// TIA Portal V20 export
FUNCTION_BLOCK "FB_HmiKeysSignalsManu"   // FB813, SCL
{ S7_Optimized_Access := 'TRUE' }
// stored: AutoNumber false, MemoryReserve 100, SetENOAutomatically false
   VAR_IN_OUT
      ioOPC : "UDT_OPC_Button";
   END_VAR
   VAR
      sKeySWStatus : Bool;
      sKeySWToggleStatus : Bool;
      sKeyDisable : Bool;
      sKeySWPositiveFront : Bool;
      sKeySWNegativeFront : Bool;
      sKeySWTogglePositiveFront : Bool;
      sKeySWToggleNegativeFront : Bool;
      sLedSWStatus : Bool;
      sLedSWStatusBlink : Bool;
      sRT_KeySWPositiveFront { S7_SetPoint := 'True'} : R_TRIG;
      sFT_KeySWNegativeFront { S7_SetPoint := 'True'} : F_TRIG;
      sRT_KeySWTogglePositiveFront { S7_SetPoint := 'True'} : R_TRIG;
      sFT_KeySWToggleNegativeFront { S7_SetPoint := 'True'} : F_TRIG;
   END_VAR
BEGIN
   REGION Description header 
       //==================================================================================
       // POSALUX Swiss SA / (C) Copyright 2025
       //----------------------------------------------------------------------------------
       // Title: FB_HmiKeysSignalsManu 
       // Comment/Function: 
       //
       // Author: Fabien Waldt
       // Engineering: TIA Portal v19
       //----------------------------------------------------------------------------------
       // Change log table:
       // Version  | Date     | Expert in charge | Changes applied
       // ---------|----------|------------------|------------------------------------
       // 00.00.01 | 20250911 | WFA              | First released version
       // ==================================================================================
   END_REGION

   REGION Key Enable
       #ioOPC.bEnable := NOT #sKeyDisable;
   END_REGION

   REGION Inputs keys
           // Management of the software input
           IF NOT #sKeyDisable THEN
               #sKeySWStatus := #ioOPC.bClick;
           // ELSE
           //     #sKeySWStatus := FALSE;
           //     #sKeySWToggleStatus := FALSE;
           END_IF;

           // Reset KeyOPCStatus (bClick from HMI)
           #ioOPC.bClick := FALSE;

           // Rising/falling edge detection when pressing the button
           #sRT_KeySWPositiveFront(CLK := #sKeySWStatus,
                                  Q => #sKeySWPositiveFront);

           #sFT_KeySWNegativeFront(CLK := #sKeySWStatus,
                                  Q => #sKeySWNegativeFront);

           // Toggle state update
           IF #sKeySWPositiveFront  THEN
               #sKeySWToggleStatus := NOT #sKeySWToggleStatus;
           END_IF;

           // Rising/falling edge detection of the toggle state
           #sRT_KeySWTogglePositiveFront(CLK := #sKeySWToggleStatus,
                                        Q => #sKeySWTogglePositiveFront);

           #sFT_KeySWToggleNegativeFront(CLK := #sKeySWToggleStatus,
                                        Q => #sKeySWToggleNegativeFront);
   END_REGION

   REGION Outputs LED   
       #ioOPC.bIsPressed := TRUE;

       // On / Off Status
       IF #sLedSWStatus THEN
           #ioOPC.eColor := 2;
       ELSE
           #ioOPC.eColor := 0;
       END_IF;

       // Blink Status
       #ioOPC.bBlink := #sLedSWStatusBlink;
   END_REGION
END_FUNCTION_BLOCK
